TYPE E_InstrumentType :
(
	InstruType_UNKNOWM := 0,
	InstruType_endoscope := 1,
	InstruType_NeedleGripper := 2,
	InstruType_Energy :=3
);
END_TYPE

(* stored: Version 1.1.0.1, ProductVersion 3.1.4024.12
   DUT E_InstrumentType: Id {d0857a03-19bb-4ed9-915e-05d1b2d79b50} *)
